// TIA Portal V19 export
TYPE "lexchangetray_typeUnEmn_toHandlingXyzDeliver"
// Type: lexchangetray_typeUnEmn_toHandlingXyzReq
// Type: lexchangetray_typeUnEmn_toHandlingXyzFeedback
// stored: Access Published
   STRUCT
      feedback : "lexchangetray_typeUnEmn_toHandlingXyzFeedback";
      req : "lexchangetray_typeUnEmn_toHandlingXyzReq";
   END_STRUCT;
END_TYPE
